{attribute 'qualified_only'}
{attribute 'strict'}
TYPE E_AssyState :
(
	PASS := 0,
	FAIL := 1,
	BREAK := 2
);
END_TYPE

(* stored: Version 1.1.0.1
   DUT E_AssyState: Id {dd1be568-d0e6-0f7e-3fed-0f598f5b6768} *)
